INTERFACE ITcoTask EXTENDS ITcoObject, ITcoRestorable

METHOD Abort
END_METHOD

PROPERTY Busy : BOOL
GET
END_GET
END_PROPERTY

PROPERTY Done : BOOL
GET
END_GET
END_PROPERTY

PROPERTY Error : BOOL
GET
END_GET
END_PROPERTY

(*~
	<docu>
		<summary>
			Use to start the execution of the task. The starting is possible from Ready state.
			<para>Moreover it is also possible to start the task again from Done state by performing the '''rising edge''' of the calling of the Invoke() method.</para>
			<p>Analogously to the xExecute signal of the <a href="https://plcopen.org/sites/default/files/downloads/creating_plcopen_compliant_function_block_libraries.pdf" title="Title"> PLCopen </a> motion function blocks.</p>
		</summary>
	</docu>
~*)
METHOD Invoke : ITcoTaskStatus
END_METHOD

END_INTERFACE

(* stored: Version 1.1.0.1
   Itf ITcoTask: Id {cac22837-decb-473a-90cc-a2a0eb0af979}
   Method Abort: Id {bd5ab69c-680d-4a5f-8d60-e0b5a722eb53}
   Property Busy: Id {0129cc85-1c85-4e79-9ded-86385e7537c6}
   Get Get: Id {ee3882a2-93e4-41cb-a89a-ea0695c17523}
   Property Done: Id {861ae878-400c-424e-8d3b-d7fd3d0b3027}
   Get Get: Id {64ee82f5-904a-4dc9-a108-2cc4256f4501}
   Property Error: Id {122a6517-d02a-4727-8caf-901f14e4e756}
   Get Get: Id {6535ce5e-74bd-4116-b8ac-4db07f7e5bea}
   Method Invoke: Id {39057362-a416-01a7-33c7-5986432fcedd} *)
